INTERFACE I_BaseMotionStage

METHOD CalibrateEncoderValue
VAR_INPUT
END_VAR
END_METHOD

METHOD DriveVirtual
VAR_INPUT
END_VAR
END_METHOD

METHOD ExposeNCParams
VAR_INPUT
END_VAR
END_METHOD

METHOD Homing
VAR_INPUT
END_VAR
END_METHOD

METHOD LogErrors
VAR_INPUT
END_VAR
END_METHOD

METHOD Processing
VAR_INPUT
END_VAR
END_METHOD

END_INTERFACE

(* stored: Version 1.1.0.1
   Itf I_BaseMotionStage: Id {9d77220c-57f1-4b48-a9ff-431bdfa81569}
   Method CalibrateEncoderValue: Id {eb078641-c453-45be-aaf5-1b7eee891909}
   Method DriveVirtual: Id {c948913d-1fe0-49a4-a017-d0eddeea2ec5}
   Method ExposeNCParams: Id {14c2064d-4177-4ca1-a486-0df861004639}
   Method Homing: Id {51dac488-4eeb-4e68-ac46-f008cc53f888}
   Method LogErrors: Id {bf350395-4325-4d9e-8461-b7950ba3f1be}
   Method Processing: Id {b47f0e8c-91a2-42aa-96ef-aeaf8d3990f7} *)
